# EPICS IOC start-up script: examples/test/el5032/el5032.iocsh
require ecmccfg,kiveln

${SCRIPTEXEC} ${ECMC_CONFIG_ROOT}addSlave.cmd,       "HW_DESC=EL5032, SLAVE_ID=9"

#- Reverse encoder direction 0x80p8:01:
#- ecmcConfigOrDie "Cfg.EcAddSdo(${ECMC_EC_SLAVE_NUM},0x8008,0x01,1,1)"

#- offset, we need to set 8 bytes (int64), but ECMC only supports up to 4 bytes --> TODO: create issue
#- ecmcConfigOrDie "Cfg.EcAddSdo(${ECMC_EC_SLAVE_NUM},0x8008,0x12,5000,8)"

#- switching of the supply voltage was _not_ tested.

#- #############################################################################
#- apply configuration
${SCRIPTEXEC} ${ECMC_CONFIG_ROOT}applyConfig.cmd
#- #############################################################################
#- go active
${SCRIPTEXEC} ${ECMC_CONFIG_ROOT}setAppMode.cmd

#- reset all errors
ecmcConfigOrDie "ControllerErrorReset()"
